FUNCTION_BLOCK FB_Licht
VAR_INPUT
	bEinKurz				: BOOL;
	bEinLang				: BOOL;
	bAus 						: BOOL;
	tKurz						: TIME := t#5m;
	tLang 					: TIME := t#60m;
END_VAR
VAR_OUTPUT
END_VAR
VAR_IN_OUT
	bGruppeAus : BOOL;
END_VAR
VAR
	bInit 			: BOOL := TRUE;
	bInVisu			: BOOL;
	bIn					: BOOL;

	bKlickEnable	: BOOL;
	bLangEnable		: BOOL;

	(* %I / %Q ********************)
	IbInTaster		AT %I* : BOOL;
	QbOutLicht		AT %Q* : BOOL;

	tofEin			: TOF;

	fbTaster 		: FB_Taster;

  fbLog : FB_LoggerSetMsg;
END_VAR

IF bInit THEN
	bKlickEnable := (tkurz <> t#0s);
	bLangEnable := (tLang <> t#0s);
	bInit := FALSE;
END_IF


bIn := IbInTaster OR bInVisu;
fbTaster(bIn:= bIn);

IF bKlickEnable
AND (fbTaster.bKlick
		OR bEinKurz
		OR gbLichtZentralEin)
THEN
	tofEin(IN:= TRUE, PT:= tkurz);
ELSIF bLangEnable
AND (fbTaster.bLang
		OR bEinLang)
THEN
	tofEin(IN:= TRUE, PT:= tLang);
END_IF
tofEin(IN:= FALSE);

IF fbTaster.bLang AND bKlickEnable AND bLangEnable THEN
  IF NOT QbOutLicht THEN
    fbLog.M_AddMsgHint('Licht EIN Taster');
  END_IF
	QbOutLicht := TRUE;
ELSIF bEinKurz OR bEinLang THEN
  IF NOT QbOutLicht THEN
    fbLog.M_AddMsgHint('Licht EIN INPUT');
  END_IF
	QbOutLicht := TRUE;
ELSIF gbLichtZentralEin THEN
	QbOutLicht := TRUE;
  //fbLog.M_AddMsgHint('Licht EIN ZentralEin');
END_IF

IF (fbTaster.bKlick
		AND bKlickEnable)
OR (fbTaster.bLang
		AND NOT bKlickEnable
		AND bLangEnable)
THEN
  IF NOT QbOutLicht THEN
    IF NOT QbOutLicht THEN
      fbLog.M_AddMsgHint('Licht EIN Taster');
    END_IF
  	QbOutLicht := TRUE;
  ELSE
    IF QbOutLicht THEN
      fbLog.M_AddMsgHint('Licht AUS Taster');
    END_IF
  	QbOutLicht := FALSE;
  END_IF
END_IF

IF QbOutLicht AND NOT tofEin.Q THEN
  IF QbOutLicht THEN
    fbLog.M_AddMsgWarning('Licht AUS Taster');
  END_IF
	QbOutLicht := FALSE;
ELSIF bAus THEN
  IF QbOutLicht THEN
    fbLog.M_AddMsgWarning('Licht AUS INPUT');
  END_IF
	QbOutLicht := FALSE;
ELSIF gbLichtZentralAus THEN
	QbOutLicht := FALSE;
  //fbLog.M_AddMsgHint('Licht AUS ZentralAus');
END_IF

IF fbTaster.bKlick2 THEN
	bGruppeAus := TRUE;
END_IF

END_FUNCTION_BLOCK

(* stored: Version 1.1.0.1, ProductVersion 3.1.4018.9
   POU FB_Licht: Id {7f37c4c1-ae20-4f41-bfff-98dfaf279b41}, SpecialFunc None *)
